SUBAPPLICATION Ventilsteuerung_Uebung_072 (* GBSD auf UT ausgeben *)
  (* Standard: 61499-2 *)
  (* Version 1.0, 2023-10-23, franz *)
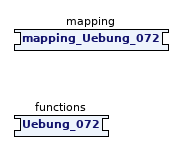
  SUBAPPS
    mapping : mapping_Uebung_072;
    functions : Uebung_072;
  END_SUBAPPS
END_SUBAPPLICATION
